// TIA Portal V17 export
// export: Created 2024-06-24T14:22:52.4686101Z, ExportSetting WithDefaults, DisplayName Totally Integrated Automation Portal, DisplayVersion V17, DisplayName TIA Portal Openness, DisplayVersion V17, DisplayName TIA Portal Version Control Interface, DisplayVersion V17, DisplayName STEP 7 Professional, DisplayVersion V17, DisplayName STEP 7 Safety, DisplayVersion V17, DisplayName WinCC Advanced, DisplayVersion V17
FUNCTION "Block_1" : Void   // FC1, LAD
{ S7_Optimized_Access := 'TRUE' }
VERSION : 0.1
// stored: AutoNumber true, IsIECCheckEnabled false, SetENOAutomatically false, UDAEnableTagReadback false
BEGIN

REGION Network 2
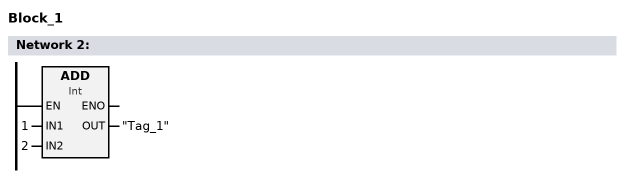
   RUNG wire#powerrail
      { S7_Templates := "SrcType := Int" } Add(in1 := 1, in2 := 2, out => "Tag_1")
   END_RUNG
   // the same network as SCL:
   "Tag_1" := 1 + 2;
END_REGION
END_FUNCTION
